(* LS Electric XG5000 project: XMC_SingleAxis_FBs *)
(* sample programs for single axis function blocks. *)
(* PLC LSPLC *)
(* module base 0 slot 0: Input/Output Module:XMC-DN24 (DC 24V Input 8Points/TR output 16Points) *)
(* module base 0 slot 1: Internal Analog Input/Output:XMF-AH04E (A/D voltage/current 2 channels, D/A voltage 2 channels) *)
(* task Periodic Task: Kind=2 *)
(* task Initialization Task: Kind=1 *)
(* task NC Program: Kind=6 *)
VAR_GLOBAL
    ContinuousRelative_INST : MC_MOVECONTINUOUSRELATIVE; (* MC_MoveContinuousRelative fb *)
    Relative_INST : MC_MOVECONTINUOUSRELATIVE; (* MC_MoveContinuousRelative fb *)
END_VAR

PROGRAM ECAT_Connect_Example (* task: Scan Program *)
VAR
    Connect_Error : BOOL; (* status that LS_Connect has an error *)
    Connect_ErrorID : WORD; (* LS_Connect Error number *)
    Connect_INST : LS_CONNECT; (* LS_Connect fb *)
    Disconnect_Error : BOOL; (* status that LS_Disconnect has an error *)
    Disconnect_ErrorID : WORD; (* Error Number for LS_Disconnect FB *)
    Disconnect_INST : LS_DISCONNECT; (* LS_Disconnect fb *)
    Execute_Connect : BOOL; (* Execute LS_Connect fb *)
    Execute_Disconnect : BOOL; (* execute LS_Disconnect fb *)
END_VAR

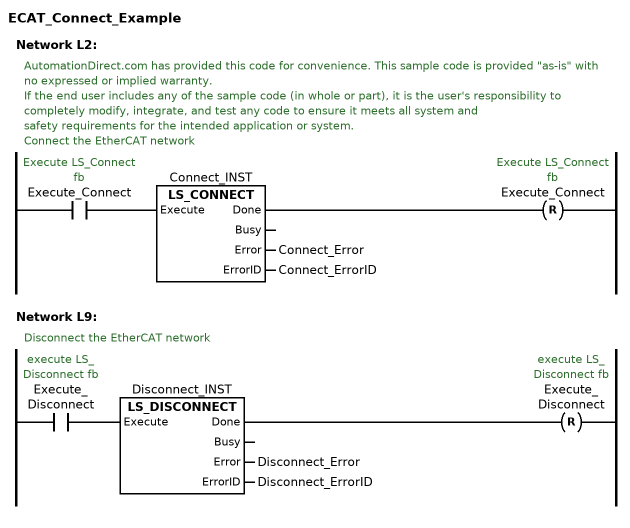
(* AutomationDirect.com has provided this code for convenience. This sample code is provided "as-is" with no expressed or implied warranty. / If the end user includes any of the sample code (in whole or part), it is the user's responsibility to completely modify, integrate, and test any code to ensure it meets all system and / safety requirements for the intended application or system. *)
(* Connect the EtherCAT network *)
(* Rung L2 *)
Connect_INST(Execute := Execute_Connect, Error => Connect_Error, ErrorID => Connect_ErrorID);
IF Connect_INST.Done THEN Execute_Connect := FALSE; END_IF;
(* Disconnect the EtherCAT network *)
(* Rung L9 *)
Disconnect_INST(Execute := Execute_Disconnect, Error => Disconnect_Error, ErrorID => Disconnect_ErrorID);
IF Disconnect_INST.Done THEN Execute_Disconnect := FALSE; END_IF;
END_PROGRAM

PROGRAM MC_Power_Example (* task: Scan Program *)
VAR
    Axis1 : UINT; (* used to tell MC function blocks to use axis 1 *)
    Axis1_MCPower_Error : BOOL; (* status of MC_Power error status *)
    Axis1_MCPower_ErrorID : WORD; (* error id of Axis 1 MC_Power *)
    Axis1_Power_Status : BOOL; (* status of axis 1 power *)
    Axis1_Power_Valid : BOOL; (* Axis1 power status is valid *)
    Power_INST : MC_POWER; (* MC_Power fb *)
    Power_On_Axis1 : BOOL; (* command to turn on power to axis 1 *)
END_VAR

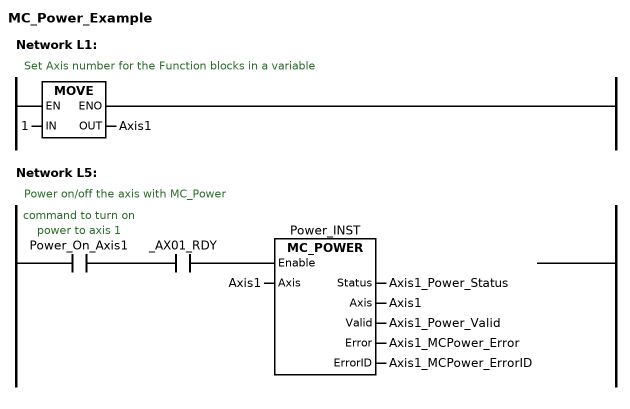
(* Set Axis number for the Function blocks in a variable *)
(* Rung L1 *)
Axis1 := 1;
(* Power on/off the axis with MC_Power *)
(* Rung L5 *)
Power_INST(Enable := Power_On_Axis1 AND _AX01_RDY, Axis := Axis1, Status => Axis1_Power_Status, Axis => Axis1, Valid => Axis1_Power_Valid, Error => Axis1_MCPower_Error, ErrorID => Axis1_MCPower_ErrorID);
END_PROGRAM

PROGRAM Home_Example (* task: Scan Program *)
(* example of MC_Home and LS_Home *)
VAR
    Axis1 : UINT; (* used to tell MC function blocks to use axis 1 *)
    Execute_LS_Home : BOOL; (* Execute LS_Home fb *)
    Execute_MC_Home : BOOL; (* execute MC_Home fb *)
    Home_INST : MC_HOME; (* MC_Home fb *)
    LSHome_Aborted : BOOL; (* LS_Home fb command aborted status *)
    LSHome_Active : BOOL; (* LS_Home fb active status *)
    LSHome_Busy : BOOL; (* LS_Home busy status *)
    LSHome_Error : BOOL; (* LSHome fb error status *)
    LSHome_ErrorID : WORD; (* LS_Home fb error id value *)
    LS_Home_INST : LS_HOME; (* LS_Home fb *)
    MCHome_Aborted : BOOL; (* MC_Home command was aborted *)
    MCHome_Active : BOOL; (* MC_Home is active *)
    MCHome_Busy : BOOL; (* MC_Home is busy *)
    MCHome_Error : BOOL; (* error status of MC_Home *)
    MCHome_ErrorID : WORD; (* error id value for MC_Home *)
END_VAR

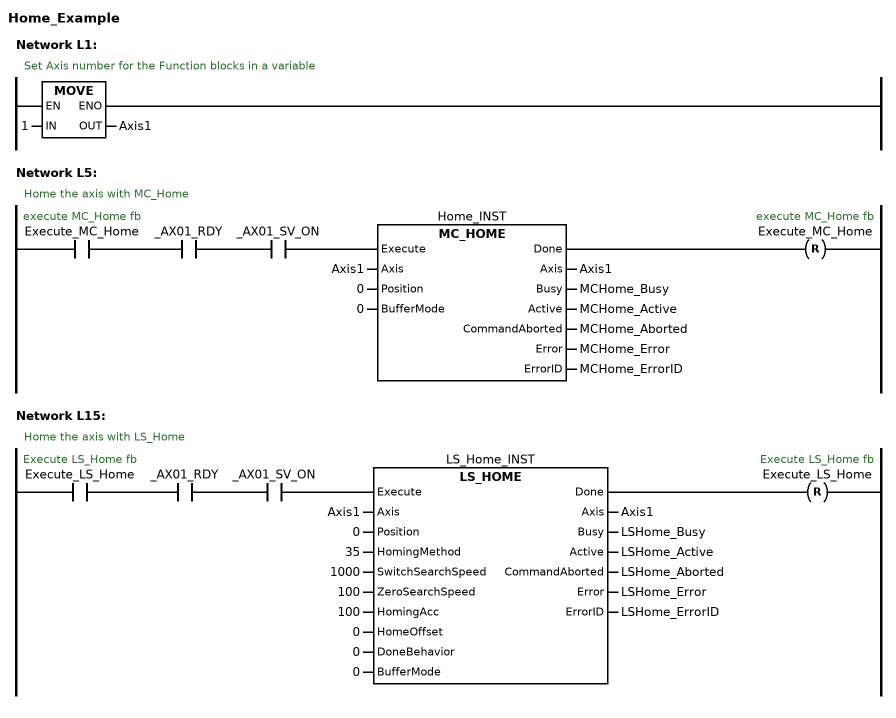
(* Set Axis number for the Function blocks in a variable *)
(* Rung L1 *)
Axis1 := 1;
(* Home the axis with MC_Home *)
(* Rung L5 *)
Home_INST(Execute := Execute_MC_Home AND _AX01_RDY AND _AX01_SV_ON, Axis := Axis1, Position := 0, BufferMode := 0, Axis => Axis1, Busy => MCHome_Busy, Active => MCHome_Active, CommandAborted => MCHome_Aborted, Error => MCHome_Error, ErrorID => MCHome_ErrorID);
IF Home_INST.Done THEN Execute_MC_Home := FALSE; END_IF;
(* Home the axis with LS_Home *)
(* Rung L15 *)
LS_Home_INST(Execute := Execute_LS_Home AND _AX01_RDY AND _AX01_SV_ON, Axis := Axis1, Position := 0, HomingMethod := 35, SwitchSearchSpeed := 1000, ZeroSearchSpeed := 100, HomingAcc := 100, HomeOffset := 0, DoneBehavior := 0, BufferMode := 0, Axis => Axis1, Busy => LSHome_Busy, Active => LSHome_Active, CommandAborted => LSHome_Aborted, Error => LSHome_Error, ErrorID => LSHome_ErrorID);
IF LS_Home_INST.Done THEN Execute_LS_Home := FALSE; END_IF;
END_PROGRAM

PROGRAM MCStop_MCHalt_Examples (* task: Scan Program *)
(* Examples of MC_Stop and MC_Hault function blocks. *)
VAR
    Axis1 : UINT; (* used to tell MC function blocks to use axis 1 *)
    Execute_MCHalt : BOOL; (* execute MC_Halt FB *)
    Execute_MCStop : BOOL; (* command to execute MC_Stop fb *)
    MCHalt_Aborted : BOOL; (* MC_Hault command aborted status *)
    MCHalt_Active : BOOL; (* MC_Halt active status *)
    MCHalt_Busy : BOOL; (* Busy status for MC_Halt *)
    MCHalt_Error : BOOL; (* MC_Halt error status *)
    MCHalt_ErrorID : WORD; (* MC_Halt Error identification value *)
    MCHalt_INST : MC_HALT; (* MC_Halt function block *)
    MCStop_Aborted : BOOL; (* MC_Stop aborted status *)
    MCStop_Busy : BOOL; (* MC_Stop Busy Status *)
    MCStop_Error : BOOL; (* MC_Stop error status *)
    MCStop_ErrorID : WORD; (* MC_Stop error identification value *)
    MCStop_INST : MC_STOP; (* MC_Stop function block *)
END_VAR

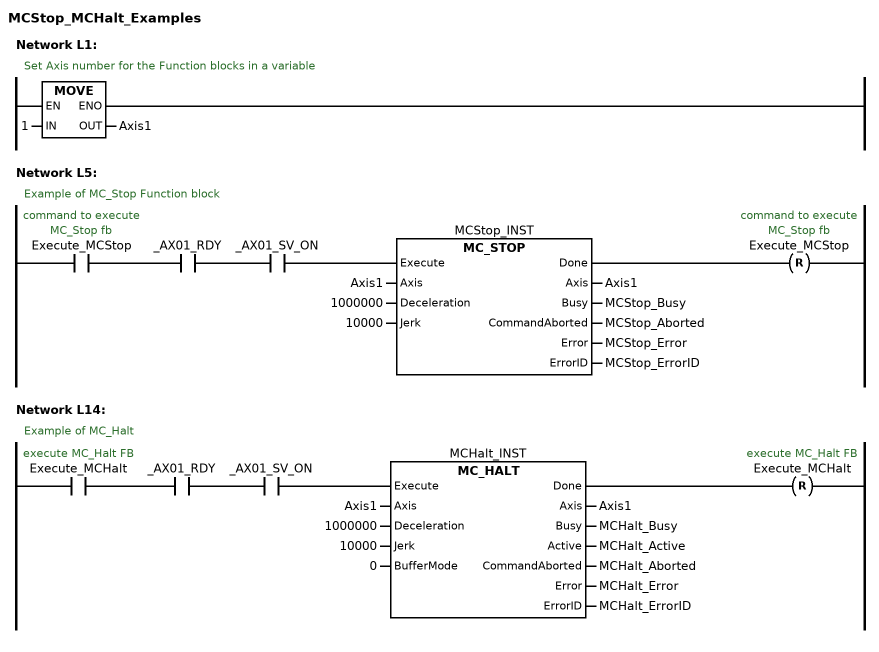
(* Set Axis number for the Function blocks in a variable *)
(* Rung L1 *)
Axis1 := 1;
(* Example of MC_Stop Function block *)
(* Rung L5 *)
MCStop_INST(Execute := Execute_MCStop AND _AX01_RDY AND _AX01_SV_ON, Axis := Axis1, Deceleration := 1000000, Jerk := 10000, Axis => Axis1, Busy => MCStop_Busy, CommandAborted => MCStop_Aborted, Error => MCStop_Error, ErrorID => MCStop_ErrorID);
IF MCStop_INST.Done THEN Execute_MCStop := FALSE; END_IF;
(* Example of MC_Halt *)
(* Rung L14 *)
MCHalt_INST(Execute := Execute_MCHalt AND _AX01_RDY AND _AX01_SV_ON, Axis := Axis1, Deceleration := 1000000, Jerk := 10000, BufferMode := 0, Axis => Axis1, Busy => MCHalt_Busy, Active => MCHalt_Active, CommandAborted => MCHalt_Aborted, Error => MCHalt_Error, ErrorID => MCHalt_ErrorID);
IF MCHalt_INST.Done THEN Execute_MCHalt := FALSE; END_IF;
END_PROGRAM

PROGRAM MC_ReadMotionInfo_Example (* task: Scan Program *)
(* example program for MC_ReadMotionInfo *)
VAR
    Axis1 : UINT; (* used to tell MC function blocks to use axis 1 *)
    Axis1_Info_Busy : BOOL; (* Axis 1 MC_ReadMotionInfo is busy *)
    Axis1_Info_Error : BOOL; (* Axis 1 MC_ReadMotionInfo error status *)
    Axis1_Info_ErrorID : WORD; (* Axis 1 MC_ReadMotionInfo error identfication *)
    Axis1_Info_Valid : BOOL; (* MC_ReadMotionInfo fb for axis 1 is valid *)
    Axis1_ParameterNumber : INT; (* Parameter number for MC_ReadMotionInfo *)
    Axis1_Value32 : REAL; (* Axis 1 MC_ReadMotionInfo Value32 outptut *)
    Axis1_Value64 : LREAL; (* Axis1 MC_ReadMotionInfo Value64 output *)
    MotionInfo_INST : MC_READMOTIONINFO; (* MC_ReadMotionInfo function block *)
    Read_Axis1_MotionInfo : BOOL; (* command to read axis 1 motion information *)
END_VAR

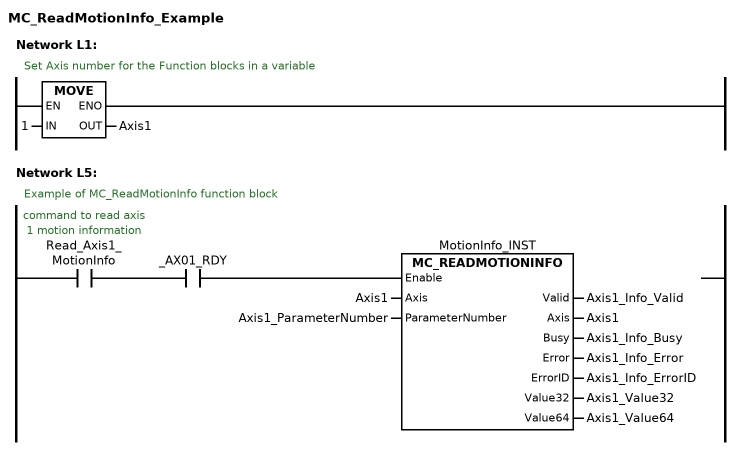
(* Set Axis number for the Function blocks in a variable *)
(* Rung L1 *)
Axis1 := 1;
(* Example of MC_ReadMotionInfo function block *)
(* Rung L5 *)
MotionInfo_INST(Enable := Read_Axis1_MotionInfo AND _AX01_RDY, Axis := Axis1, ParameterNumber := Axis1_ParameterNumber, Valid => Axis1_Info_Valid, Axis => Axis1, Busy => Axis1_Info_Busy, Error => Axis1_Info_Error, ErrorID => Axis1_Info_ErrorID, Value32 => Axis1_Value32, Value64 => Axis1_Value64);
END_PROGRAM

PROGRAM MC_ReadActualPosition_Example (* task: Scan Program *)
(* example program for MC_ReadActualPosition function block *)
VAR
    Axis1 : UINT; (* used to tell MC function blocks to use axis 1 *)
    Axis1_Position_Busy : BOOL; (* MC_ReadActualPosition is busy *)
    Axis1_Position_Error : BOOL; (* MC_ReadActualPosition error status *)
    Axis1_Position_ErrorID : WORD; (* MC_ReadActualPosition error identification *)
    Axis1_Position_Valid : BOOL; (* Axis 1 MC_ReadActualPosition value is valid *)
    Axis1_Position_Value32 : REAL; (* REAL value of Axis1 current position *)
    Axis1_Position_Value64 : LREAL; (* Axis 1 LREAL position value *)
    Axis1_Read_Position : BOOL; (* enable Axis1 MC_ReadActualPosition fb *)
    ReadPosition_INST : MC_READACTUALPOSITION; (* MC_ReadActualPosition function block *)
END_VAR

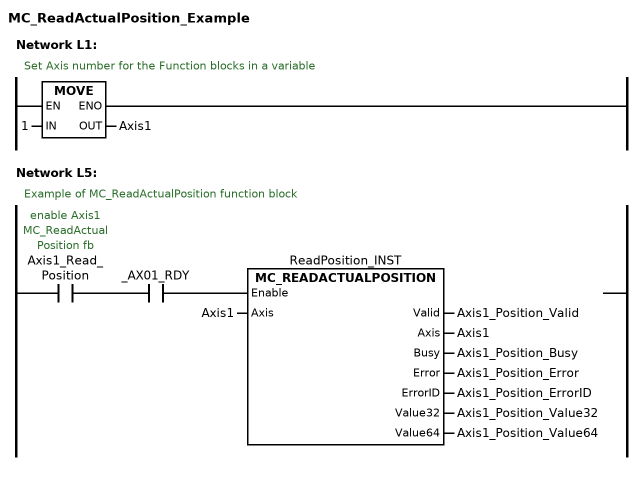
(* Set Axis number for the Function blocks in a variable *)
(* Rung L1 *)
Axis1 := 1;
(* Example of MC_ReadActualPosition function block *)
(* Rung L5 *)
ReadPosition_INST(Enable := Axis1_Read_Position AND _AX01_RDY, Axis := Axis1, Valid => Axis1_Position_Valid, Axis => Axis1, Busy => Axis1_Position_Busy, Error => Axis1_Position_Error, ErrorID => Axis1_Position_ErrorID, Value32 => Axis1_Position_Value32, Value64 => Axis1_Position_Value64);
END_PROGRAM

PROGRAM MC_ReadActualVelocity_Example (* task: Scan Program *)
(* example program for MC_ReadActualVelocity function block *)
VAR
    Axis1 : UINT; (* used to tell MC function blocks to use axis 1 *)
    Axis1_Read_Velocity : BOOL; (* command to enable MC_ReadActualVelocity *)
    Axis1_Velocity_Busy : BOOL; (* Axis 1 MC_ReadActualVelocity busy status *)
    Axis1_Velocity_Error : BOOL; (* Axis 1 MC_ReadActualVelocity error status *)
    Axis1_Velocity_ErrorID : WORD; (* Axis 1 MC_ReadActualVelocity error identification *)
    Axis1_Velocity_Valid : BOOL; (* Axis1 MC_ReadActualVelocity is valid *)
    Axis1_Velocity_Value32 : REAL; (* Axis 1 MC_ReadActualVelocity REAL value *)
    Axis1_Velocity_Value64 : LREAL; (* Axis1 MC_ReadActualVelocity LREAL value *)
    ReadVelocity_INST : MC_READACTUALVELOCITY; (* MC_ReadActualVelocity function block *)
END_VAR

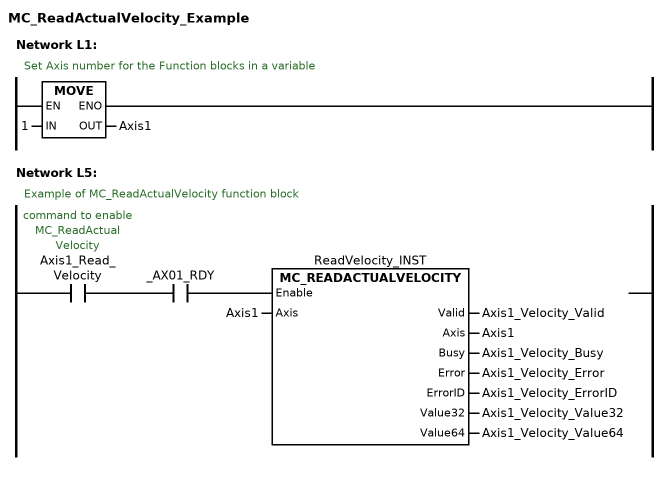
(* Set Axis number for the Function blocks in a variable *)
(* Rung L1 *)
Axis1 := 1;
(* Example of MC_ReadActualVelocity function block *)
(* Rung L5 *)
ReadVelocity_INST(Enable := Axis1_Read_Velocity AND _AX01_RDY, Axis := Axis1, Valid => Axis1_Velocity_Valid, Axis => Axis1, Busy => Axis1_Velocity_Busy, Error => Axis1_Velocity_Error, ErrorID => Axis1_Velocity_ErrorID, Value32 => Axis1_Velocity_Value32, Value64 => Axis1_Velocity_Value64);
END_PROGRAM

PROGRAM MC_ReadActualTorque_Example (* task: Scan Program *)
(* MC_ReadActualTorque function block example *)
VAR
    Axis1 : UINT; (* used to tell MC function blocks to use axis 1 *)
    Axis1_Read_Torque : BOOL; (* enable MC_ReadActualTorque *)
    Axis1_Torque_Busy : BOOL; (* Axis 1 MC_ReadActualTorque is busy *)
    Axis1_Torque_Error : BOOL; (* Axis1 MC_ReadActualTorque error status *)
    Axis1_Torque_ErrorID : WORD; (* Axis 1 MC_ReadActualTorque error identification *)
    Axis1_Torque_Valid : BOOL; (* Axis 1 MC_ReadActualTorque value is valid *)
    Axis1_Torque_Value32 : REAL; (* Axis 1 torque REAL value *)
    Axis1_Torque_Value64 : LREAL; (* Axis 1 torque LREAL value *)
    ReadTorque_INST : MC_READACTUALTORQUE; (* MC_ReadActualTorque function block *)
END_VAR

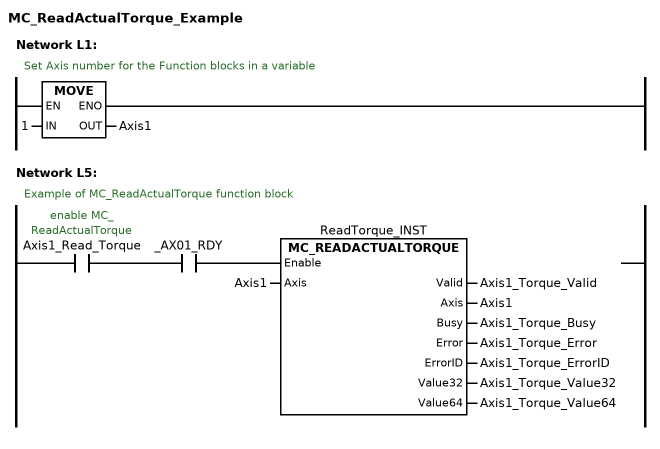
(* Set Axis number for the Function blocks in a variable *)
(* Rung L1 *)
Axis1 := 1;
(* Example of MC_ReadActualTorque function block *)
(* Rung L5 *)
ReadTorque_INST(Enable := Axis1_Read_Torque AND _AX01_RDY, Axis := Axis1, Valid => Axis1_Torque_Valid, Axis => Axis1, Busy => Axis1_Torque_Busy, Error => Axis1_Torque_Error, ErrorID => Axis1_Torque_ErrorID, Value32 => Axis1_Torque_Value32, Value64 => Axis1_Torque_Value64);
END_PROGRAM

PROGRAM MC_Reset_Example (* task: Scan Program *)
(* example of MC_Reset and MC_Reset2 function blocks. *)
VAR
    Axis1 : UINT; (* used to tell MC function blocks to use axis 1 *)
    Execute_MCReset : BOOL; (* command to execute MC_Reset FB. *)
    Execute_MCReset2 : BOOL; (* command to execute MC_Reset2 *)
    Reset1_Busy : BOOL; (* MC_Reset busy status *)
    Reset1_Error : BOOL; (* MC_Reset Error status *)
    Reset1_ErrorID : WORD; (* MC_Reset error identification *)
    Reset1_ErrorType : BOOL; (* error type for MC_Reset *)
    Reset1_INST : MC_RESET; (* MC_Reset function block *)
    Reset2_Busy : BOOL; (* busy status for MC_Reset2 *)
    Reset2_Error : BOOL; (* error status for MC_Reset2 *)
    Reset2_ErrorID : WORD; (* MC_Reset2 error identification *)
    Reset2_ErrorType : UINT; (* error type for MC_Reset2 *)
    Reset2_INST : MC_RESET2; (* MC_Reset2 function block *)
END_VAR

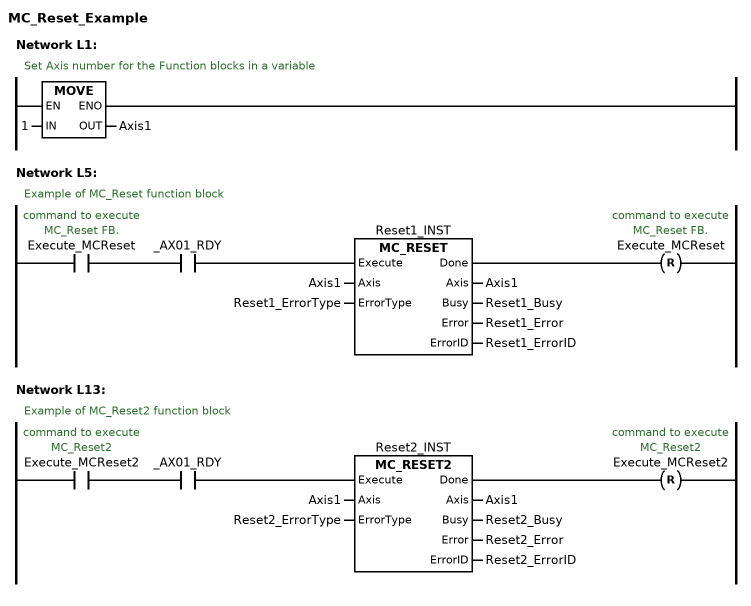
(* Set Axis number for the Function blocks in a variable *)
(* Rung L1 *)
Axis1 := 1;
(* Example of MC_Reset function block *)
(* Rung L5 *)
Reset1_INST(Execute := Execute_MCReset AND _AX01_RDY, Axis := Axis1, ErrorType := Reset1_ErrorType, Axis => Axis1, Busy => Reset1_Busy, Error => Reset1_Error, ErrorID => Reset1_ErrorID);
IF Reset1_INST.Done THEN Execute_MCReset := FALSE; END_IF;
(* Example of MC_Reset2 function block *)
(* Rung L13 *)
Reset2_INST(Execute := Execute_MCReset2 AND _AX01_RDY, Axis := Axis1, ErrorType := Reset2_ErrorType, Axis => Axis1, Busy => Reset2_Busy, Error => Reset2_Error, ErrorID => Reset2_ErrorID);
IF Reset2_INST.Done THEN Execute_MCReset2 := FALSE; END_IF;
END_PROGRAM

PROGRAM MC_MoveAbsolute_Example (* task: Scan Program *)
(* example program for MC_MoveAbsolute function block *)
VAR
    AbsoluteMove_Aborted : BOOL; (* MC_MoveAbsolute was aborted. *)
    AbsoluteMove_Acceleration : LREAL; (* acceleration for MC_MoveAbsolute *)
    AbsoluteMove_Active : BOOL; (* MC_MoveAbsolute is active *)
    AbsoluteMove_Busy : BOOL; (* MC_MoveAbsolute busy status *)
    AbsoluteMove_ContinuousUpdate : BOOL; (* continuous update status for MC_MoveAbsolute *)
    AbsoluteMove_Deceleration : LREAL; (* deceleration for MC_MoveAbsolute *)
    AbsoluteMove_Direction : UINT; (* direction of MC_MoveAbsolute *)
    AbsoluteMove_Error : BOOL; (* MC_MoveAbsolute error status *)
    AbsoluteMove_ErrorID : WORD; (* MC_MoveAbsolute error identification *)
    AbsoluteMove_Jerk : LREAL; (* jerk value for MC_MoveAbsolute *)
    AbsoluteMove_TargetPosition : LREAL; (* target position for MC_MoveAbsolute *)
    AbsoluteMove_Velocity : LREAL; (* velocity for MC_MoveAbsolute *)
    Absolute_INST : MC_MOVEABSOLUTE; (* MC_MoveAbsolute function block *)
    Axis1 : UINT; (* used to tell MC function blocks to use axis 1 *)
    Execute_Absolute_Move : BOOL; (* execute MC_MoveAbsolute function block *)
END_VAR

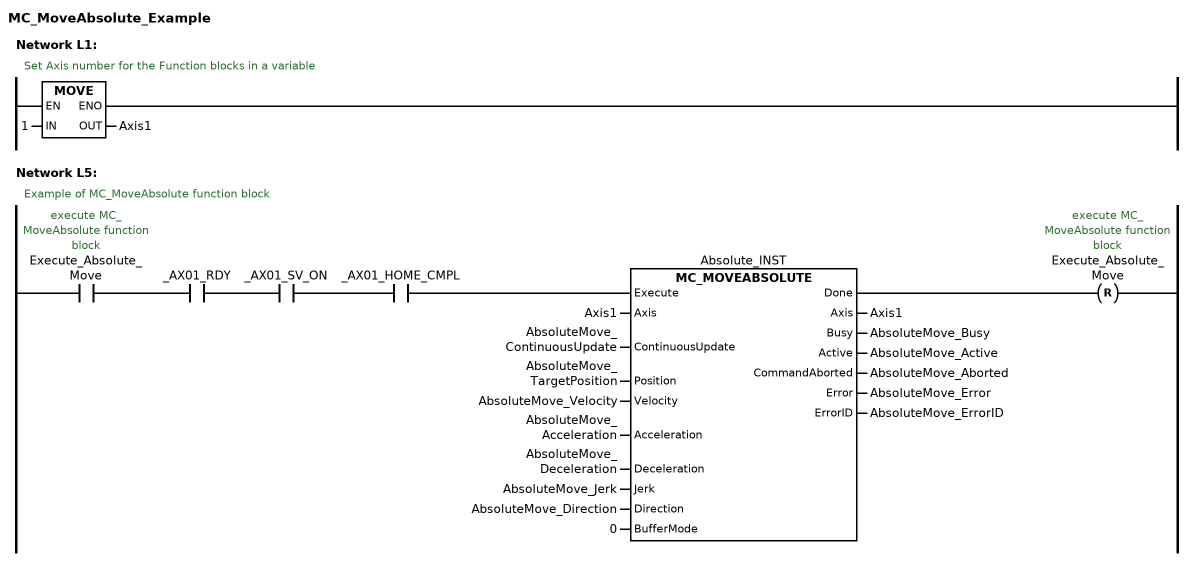
(* Set Axis number for the Function blocks in a variable *)
(* Rung L1 *)
Axis1 := 1;
(* Example of MC_MoveAbsolute function block *)
(* Rung L5 *)
Absolute_INST(Execute := Execute_Absolute_Move AND _AX01_RDY AND _AX01_SV_ON AND _AX01_HOME_CMPL, Axis := Axis1, ContinuousUpdate := AbsoluteMove_ContinuousUpdate, Position := AbsoluteMove_TargetPosition, Velocity := AbsoluteMove_Velocity, Acceleration := AbsoluteMove_Acceleration, Deceleration := AbsoluteMove_Deceleration, Jerk := AbsoluteMove_Jerk, Direction := AbsoluteMove_Direction, BufferMode := 0, Axis => Axis1, Busy => AbsoluteMove_Busy, Active => AbsoluteMove_Active, CommandAborted => AbsoluteMove_Aborted, Error => AbsoluteMove_Error, ErrorID => AbsoluteMove_ErrorID);
IF Absolute_INST.Done THEN Execute_Absolute_Move := FALSE; END_IF;
END_PROGRAM

PROGRAM MC_MoveRelative_Example (* task: Scan Program *)
(* example program for MC_MoveRelative funciton block *)
VAR
    Axis1 : UINT; (* used to tell MC function blocks to use axis 1 *)
    Execute_RelativeMove : BOOL; (* execute MC_MoveRelative *)
    RelativeMove_Aborted : BOOL; (* MC_MoveRelative aborted status *)
    RelativeMove_Acceleration : LREAL; (* acceleration for relative move *)
    RelativeMove_Active : BOOL; (* MC_MoveRelative active status *)
    RelativeMove_Busy : BOOL; (* MC_MoveRelative busy status *)
    RelativeMove_ContinuousUpdate : BOOL; (* MC_MoveRelative continuous update *)
    RelativeMove_Deceleration : LREAL; (* deceleration for relative move *)
    RelativeMove_Distance : LREAL; (* Distance for the MC_MoveRelative to move *)
    RelativeMove_Error : BOOL; (* MC_MoveRelative error status *)
    RelativeMove_ErrorID : WORD; (* MC_MoveRelative error identification *)
    RelativeMove_INST : MC_MOVERELATIVE; (* MC_MoveRelative function block *)
    RelativeMove_Jerk : LREAL; (* jerk value for relative move *)
    RelativeMove_Velocity : LREAL; (* velocity for relative move *)
END_VAR

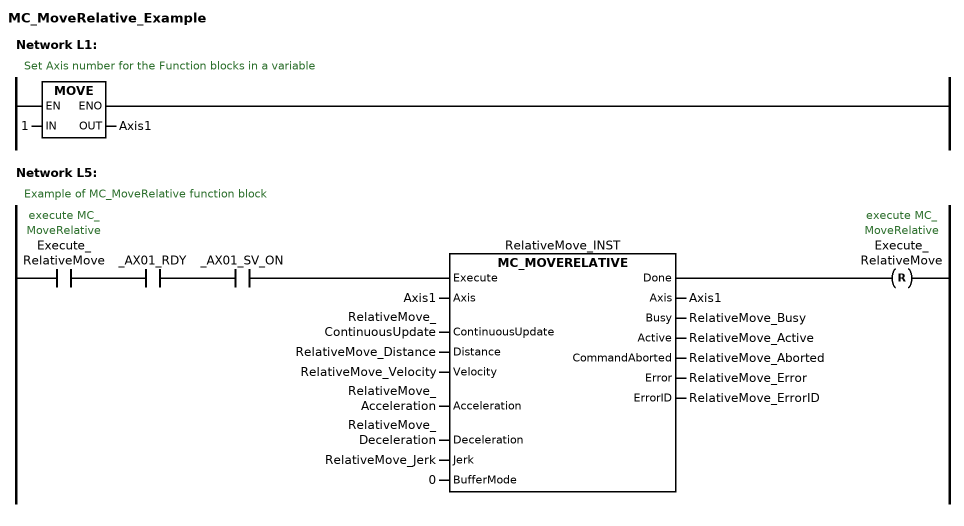
(* Set Axis number for the Function blocks in a variable *)
(* Rung L1 *)
Axis1 := 1;
(* Example of MC_MoveRelative function block *)
(* Rung L5 *)
RelativeMove_INST(Execute := Execute_RelativeMove AND _AX01_RDY AND _AX01_SV_ON, Axis := Axis1, ContinuousUpdate := RelativeMove_ContinuousUpdate, Distance := RelativeMove_Distance, Velocity := RelativeMove_Velocity, Acceleration := RelativeMove_Acceleration, Deceleration := RelativeMove_Deceleration, Jerk := RelativeMove_Jerk, BufferMode := 0, Axis => Axis1, Busy => RelativeMove_Busy, Active => RelativeMove_Active, CommandAborted => RelativeMove_Aborted, Error => RelativeMove_Error, ErrorID => RelativeMove_ErrorID);
IF RelativeMove_INST.Done THEN Execute_RelativeMove := FALSE; END_IF;
END_PROGRAM

PROGRAM MC_MoveAdditive_Example (* task: Scan Program *)
(* example program for MC_MoveAdditive *)
VAR
    AdditiveMove_Aborted : BOOL; (* MC_MoveAdditive aborted status *)
    AdditiveMove_Acceleration : LREAL; (* acceleration for MC_AdditiveMove *)
    AdditiveMove_Active : BOOL; (* MC_MoveAdditive active status *)
    AdditiveMove_Busy : BOOL; (* MC_MoveAdditive busy status *)
    AdditiveMove_ContinuousUpdate : BOOL; (* ContinuousUpdate for MC_MoveAdditive *)
    AdditiveMove_Deceleration : LREAL; (* deceleration for MC_AdditiveMove *)
    AdditiveMove_Distance : LREAL; (* distance for MC_MoveAdditive *)
    AdditiveMove_Error : BOOL; (* MC_MoveAdditive error status *)
    AdditiveMove_ErrorID : WORD; (* MC_MoveAdditive error identification *)
    AdditiveMove_INST : MC_MOVEADDITIVE; (* MC_MoveAdditive function block *)
    AdditiveMove_Jerk : LREAL; (* jerk value for MC_MoveAdditive *)
    AdditiveMove_Velocity : LREAL; (* velocity for the MC_MoveAdditive *)
    Axis1 : UINT; (* used to tell MC function blocks to use axis 1 *)
    Execute_AdditiveMove : BOOL; (* execute MC_MoveRelative *)
END_VAR

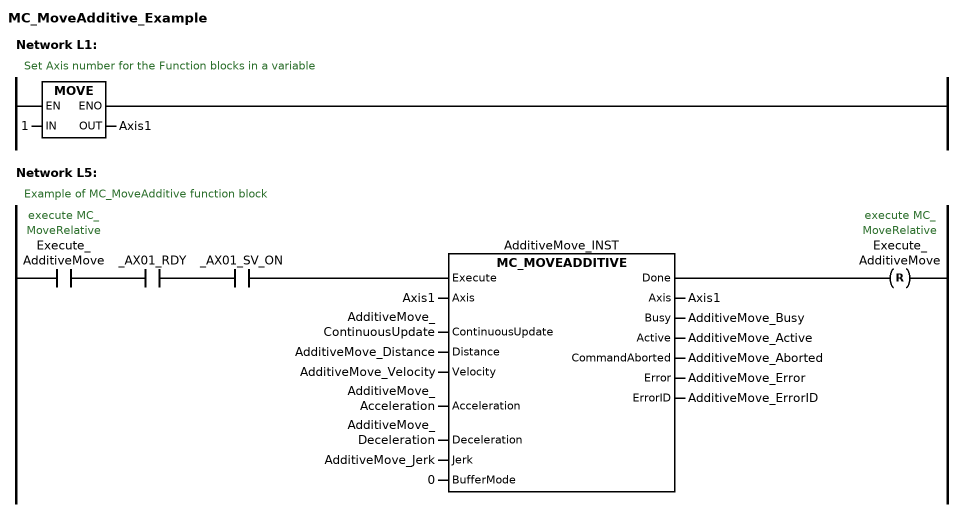
(* Set Axis number for the Function blocks in a variable *)
(* Rung L1 *)
Axis1 := 1;
(* Example of MC_MoveAdditive function block *)
(* Rung L5 *)
AdditiveMove_INST(Execute := Execute_AdditiveMove AND _AX01_RDY AND _AX01_SV_ON, Axis := Axis1, ContinuousUpdate := AdditiveMove_ContinuousUpdate, Distance := AdditiveMove_Distance, Velocity := AdditiveMove_Velocity, Acceleration := AdditiveMove_Acceleration, Deceleration := AdditiveMove_Deceleration, Jerk := AdditiveMove_Jerk, BufferMode := 0, Axis => Axis1, Busy => AdditiveMove_Busy, Active => AdditiveMove_Active, CommandAborted => AdditiveMove_Aborted, Error => AdditiveMove_Error, ErrorID => AdditiveMove_ErrorID);
IF AdditiveMove_INST.Done THEN Execute_AdditiveMove := FALSE; END_IF;
END_PROGRAM

PROGRAM MC_MoveVelocity_Example (* task: Scan Program *)
(* Example program for MC_MoveVelocity function block *)
VAR
    Axis1 : UINT; (* used to tell MC function blocks to use axis 1 *)
    Execute_MoveVelocity : BOOL; (* execute the MC_MoveVelocity Function block *)
    VelocityMove_Aborted : BOOL; (* MC_MoveVelocity Status aborted *)
    VelocityMove_Acceleration : LREAL; (* acceleration value for axis 1 MC_MoveVelocity *)
    VelocityMove_Active : BOOL; (* active status of MC_MoveVelocity *)
    VelocityMove_Busy : BOOL; (* busy status of MC_MoveVelocity *)
    VelocityMove_ContinuousUpdate : BOOL; (* setting the continuous update *)
    VelocityMove_Deceleration : LREAL; (* Axis1 deceleration value *)
    VelocityMove_Direction : UINT; (* direction of Axis 1 MC_MoveVelocity *)
    VelocityMove_Error : BOOL; (* Error status of MC_MoveVelocity *)
    VelocityMove_ErrorID : WORD; (* MC_MoveVelocity error identification *)
    VelocityMove_Jerk : LREAL; (* jerk value for axis 1 *)
    VelocityMove_Velocity : LREAL; (* velocity for Axis1 *)
    Velocity_INST : MC_MOVEVELOCITY; (* MC_MoveVelocity function block instance *)
END_VAR

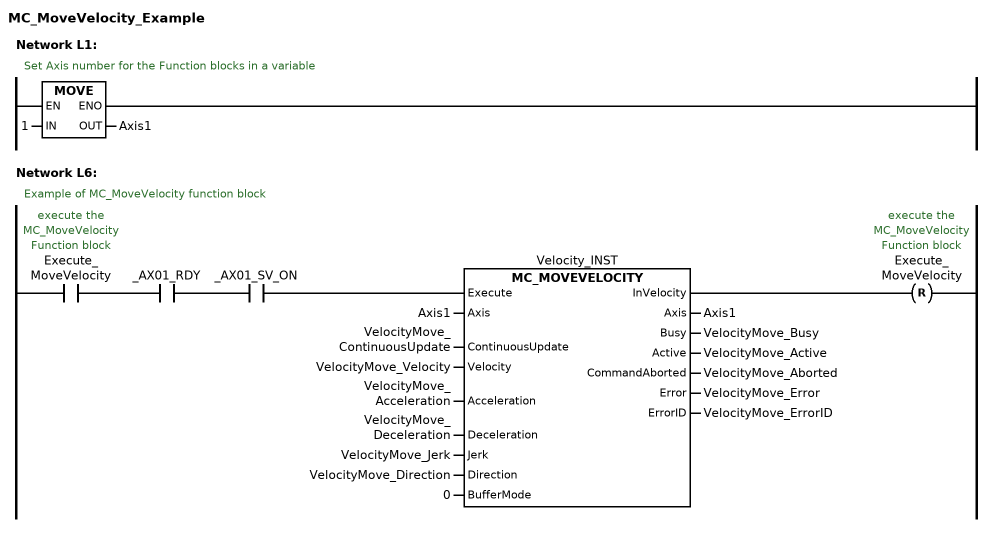
(* Set Axis number for the Function blocks in a variable *)
(* Rung L1 *)
Axis1 := 1;
(* Example of MC_MoveVelocity function block *)
(* Rung L6 *)
Velocity_INST(Execute := Execute_MoveVelocity AND _AX01_RDY AND _AX01_SV_ON, Axis := Axis1, ContinuousUpdate := VelocityMove_ContinuousUpdate, Velocity := VelocityMove_Velocity, Acceleration := VelocityMove_Acceleration, Deceleration := VelocityMove_Deceleration, Jerk := VelocityMove_Jerk, Direction := VelocityMove_Direction, BufferMode := 0, Axis => Axis1, Busy => VelocityMove_Busy, Active => VelocityMove_Active, CommandAborted => VelocityMove_Aborted, Error => VelocityMove_Error, ErrorID => VelocityMove_ErrorID);
IF Velocity_INST.InVelocity THEN Execute_MoveVelocity := FALSE; END_IF;
END_PROGRAM

PROGRAM MC_MoveContinuousAbsolute_Example (* task: Scan Program *)
(* example program for MC_MoveContinuousAbsolute function block *)
VAR
    Axis1 : UINT; (* used to tell MC function blocks to use axis 1 *)
    ContinuousAbsolute_Aborted : BOOL; (* aborted status of the function block *)
    ContinuousAbsolute_Acceleration : LREAL; (* acceleration for movement *)
    ContinuousAbsolute_Active : BOOL; (* active status of function block *)
    ContinuousAbsolute_Busy : BOOL; (* busy status *)
    ContinuousAbsolute_ContinuousUpdate : BOOL; (* MC_MoveContinuousAbsolute continuous update input *)
    ContinuousAbsolute_Deceleration : LREAL; (* deceleration for moves *)
    ContinuousAbsolute_Direction : UINT; (* direction of the movement *)
    ContinuousAbsolute_EndVelocity : LREAL; (* end velocity for MC_MoveContinuousAbsolute function block *)
    ContinuousAbsolute_Error : BOOL; (* error status of the function block *)
    ContinuousAbsolute_ErrorID : WORD; (* error identification of the function block *)
    ContinuousAbsolute_INST : MC_MOVECONTINUOUSABSOLUTE; (* MC_MoveContinuousAbsolute function block *)
    ContinuousAbsolute_Jerk : LREAL; (* jerk value for movement *)
    ContinuousAbsolute_Position : LREAL; (* target position before continuous motion *)
    ContinuousAbsolute_Velocity : LREAL; (* velocity of the absolute motion portion *)
    Execute_MoveContinuousAbsolute : BOOL; (* execute MC_MoveContinuousAbsolute *)
END_VAR

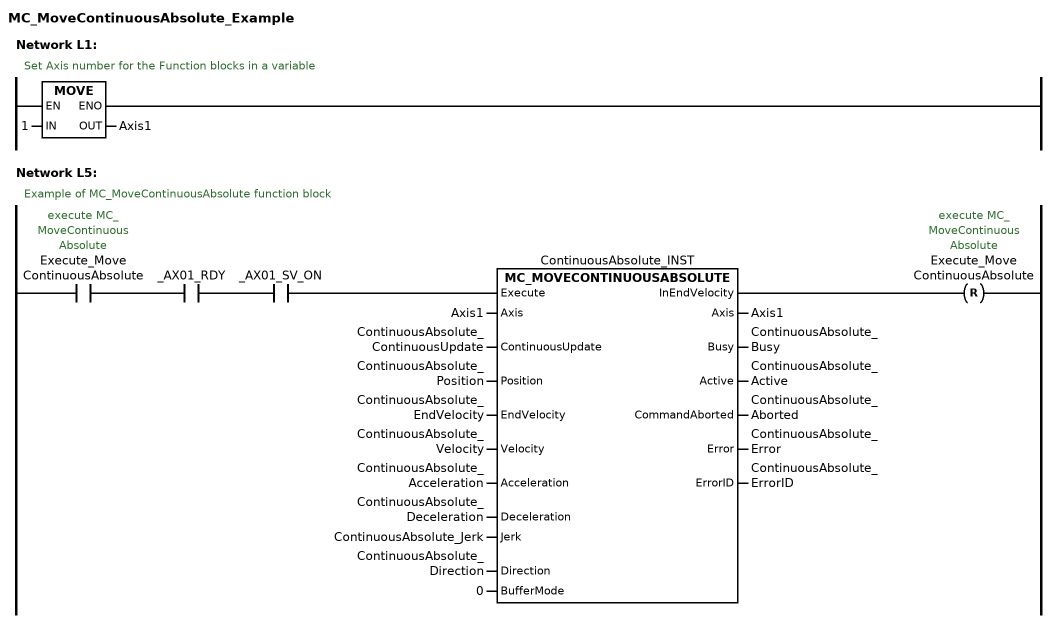
(* Set Axis number for the Function blocks in a variable *)
(* Rung L1 *)
Axis1 := 1;
(* Example of MC_MoveContinuousAbsolute function block *)
(* Rung L5 *)
ContinuousAbsolute_INST(Execute := Execute_MoveContinuousAbsolute AND _AX01_RDY AND _AX01_SV_ON, Axis := Axis1, ContinuousUpdate := ContinuousAbsolute_ContinuousUpdate, Position := ContinuousAbsolute_Position, EndVelocity := ContinuousAbsolute_EndVelocity, Velocity := ContinuousAbsolute_Velocity, Acceleration := ContinuousAbsolute_Acceleration, Deceleration := ContinuousAbsolute_Deceleration, Jerk := ContinuousAbsolute_Jerk, Direction := ContinuousAbsolute_Direction, BufferMode := 0, Axis => Axis1, Busy => ContinuousAbsolute_Busy, Active => ContinuousAbsolute_Active, CommandAborted => ContinuousAbsolute_Aborted, Error => ContinuousAbsolute_Error, ErrorID => ContinuousAbsolute_ErrorID);
IF ContinuousAbsolute_INST.InEndVelocity THEN Execute_MoveContinuousAbsolute := FALSE; END_IF;
END_PROGRAM

PROGRAM MC_MoveContinuousRelative_Example (* task: Scan Program *)
(* example of MC_MoveContinuousRelative function block *)
VAR
    Axis1 : UINT; (* used to tell MC function blocks to use axis 1 *)
    ContinuousRelative_Aborted : BOOL; (* aborted status for fb *)
    ContinuousRelative_Acceleration : LREAL; (* Acceleration for fb *)
    ContinuousRelative_Active : BOOL; (* active status for fb *)
    ContinuousRelative_Busy : BOOL; (* busy status for fb *)
    ContinuousRelative_ContinuousUpdate : BOOL; (* MC_MoveContinuousRelative update input *)
    ContinuousRelative_Deceleration : LREAL; (* deceleration for fb *)
    ContinuousRelative_Distance : LREAL; (* distance value for MC_MoveContinuousRelative *)
    ContinuousRelative_EndVelocity : LREAL; (* end velocity value for MC_MoveContinuousRelative fb *)
    ContinuousRelative_Error : BOOL; (* error status for fb *)
    ContinuousRelative_ErrorID : WORD; (* error identification for fb *)
    ContinuousRelative_Jerk : LREAL; (* Jerk value for fb *)
    ContinuousRelative_Velocity : LREAL; (* Relative move velocity for MC_MoveContinuousRelative *)
    Execute_ContinuousRelative : BOOL; (* command to execute MC_MoveContinuousRelative fb *)
END_VAR
VAR_EXTERNAL
    ContinuousRelative_INST : MC_MOVECONTINUOUSRELATIVE; (* MC_MoveContinuousRelative fb *)
END_VAR

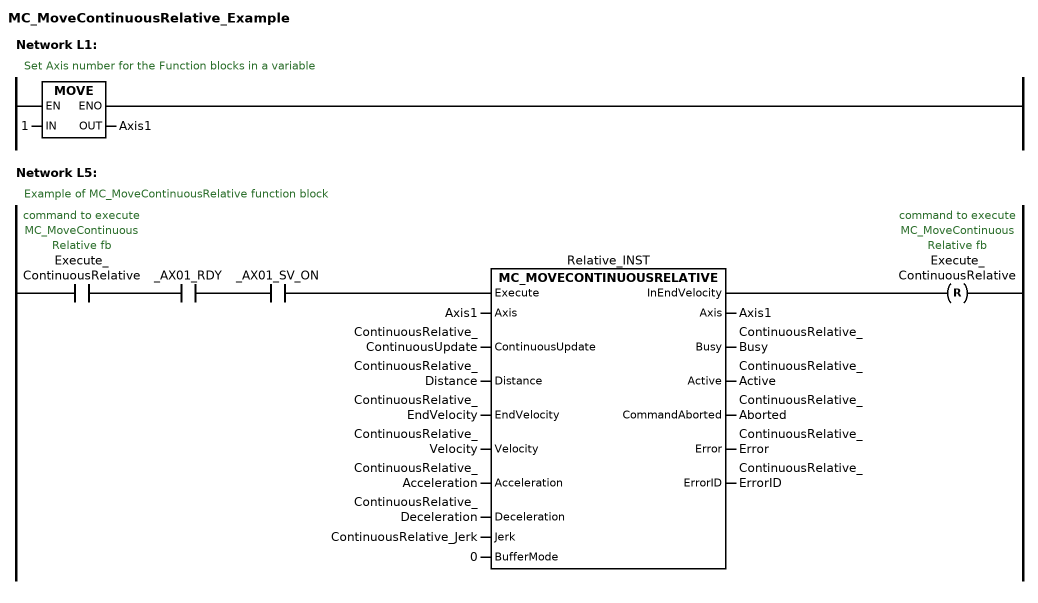
(* Set Axis number for the Function blocks in a variable *)
(* Rung L1 *)
Axis1 := 1;
(* Example of MC_MoveContinuousRelative function block *)
(* Rung L5 *)
Relative_INST(Execute := Execute_ContinuousRelative AND _AX01_RDY AND _AX01_SV_ON, Axis := Axis1, ContinuousUpdate := ContinuousRelative_ContinuousUpdate, Distance := ContinuousRelative_Distance, EndVelocity := ContinuousRelative_EndVelocity, Velocity := ContinuousRelative_Velocity, Acceleration := ContinuousRelative_Acceleration, Deceleration := ContinuousRelative_Deceleration, Jerk := ContinuousRelative_Jerk, BufferMode := 0, Axis => Axis1, Busy => ContinuousRelative_Busy, Active => ContinuousRelative_Active, CommandAborted => ContinuousRelative_Aborted, Error => ContinuousRelative_Error, ErrorID => ContinuousRelative_ErrorID);
IF Relative_INST.InEndVelocity THEN Execute_ContinuousRelative := FALSE; END_IF;
END_PROGRAM

PROGRAM MC_TorqueControl_Example (* task: Scan Program *)
(* example program for MC_TorqueControl *)
VAR
    Axis1 : UINT; (* used to tell MC function blocks to use axis 1 *)
    ContinuousUpdate : BOOL; (* continuous update of TorqueControl *)
    Execute_Torque_Control : BOOL; (* execute MC_TorqueControl function block *)
    TorqueControl_Aborted : BOOL; (* torque control aborted status *)
    TorqueControl_Active : BOOL; (* torque control active status *)
    TorqueControl_BufferMode : UINT; (* Buffer Mode for Axis 1 MC_TorqueControl *)
    TorqueControl_Busy : BOOL; (* torque control busy status *)
    TorqueControl_Direction : UINT; (* Axis1 direction for MC_TorqueControl *)
    TorqueControl_Error : BOOL; (* torque control error status *)
    TorqueControl_ErrorID : WORD; (* torque control error identification *)
    TorqueControl_TorqueRamp : LREAL; (* torque Ramp for axis 1 *)
    TorqueControl_TorqueValue : LREAL; (* torque value for axis 1 MC_TorqueControl *)
    Torque_Ctrl_INST : MC_TORQUECONTROL; (* MC_TorqueControl function block *)
END_VAR

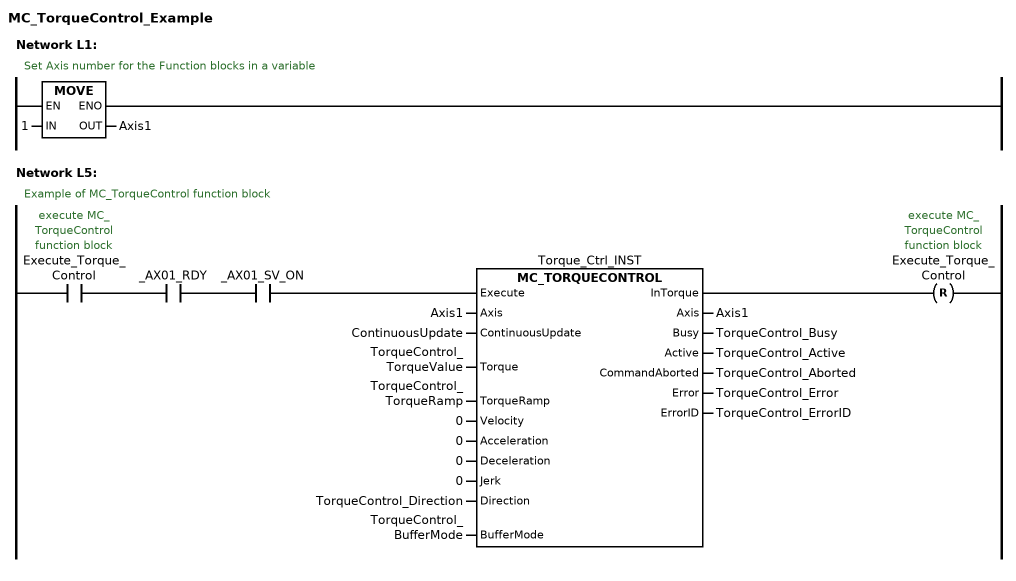
(* Set Axis number for the Function blocks in a variable *)
(* Rung L1 *)
Axis1 := 1;
(* Example of MC_TorqueControl function block *)
(* Rung L5 *)
Torque_Ctrl_INST(Execute := Execute_Torque_Control AND _AX01_RDY AND _AX01_SV_ON, Axis := Axis1, ContinuousUpdate := ContinuousUpdate, Torque := TorqueControl_TorqueValue, TorqueRamp := TorqueControl_TorqueRamp, Velocity := 0, Acceleration := 0, Deceleration := 0, Jerk := 0, Direction := TorqueControl_Direction, BufferMode := TorqueControl_BufferMode, Axis => Axis1, Busy => TorqueControl_Busy, Active => TorqueControl_Active, CommandAborted => TorqueControl_Aborted, Error => TorqueControl_Error, ErrorID => TorqueControl_ErrorID);
IF Torque_Ctrl_INST.InTorque THEN Execute_Torque_Control := FALSE; END_IF;
END_PROGRAM

PROGRAM MC_SetPosition_Example (* task: Scan Program *)
(* example of MC_SetPosition function block *)
VAR
    Axis1 : UINT; (* used to tell MC function blocks to use axis 1 *)
    Execute_Set_Position : BOOL; (* execute the MC_SetPosition FB *)
    SetPosition_Aborted : BOOL; (* aborted status of MC_SetPosition *)
    SetPosition_Busy : BOOL; (* busy status of MC_SetPosition *)
    SetPosition_Error : BOOL; (* Error status of fb *)
    SetPosition_ErrorID : WORD; (* error identification of fb *)
    SetPosition_INST : MC_SETPOSITION; (* MC_SetPosition function block *)
    SetPosition_Position : LREAL; (* position value for set position *)
END_VAR

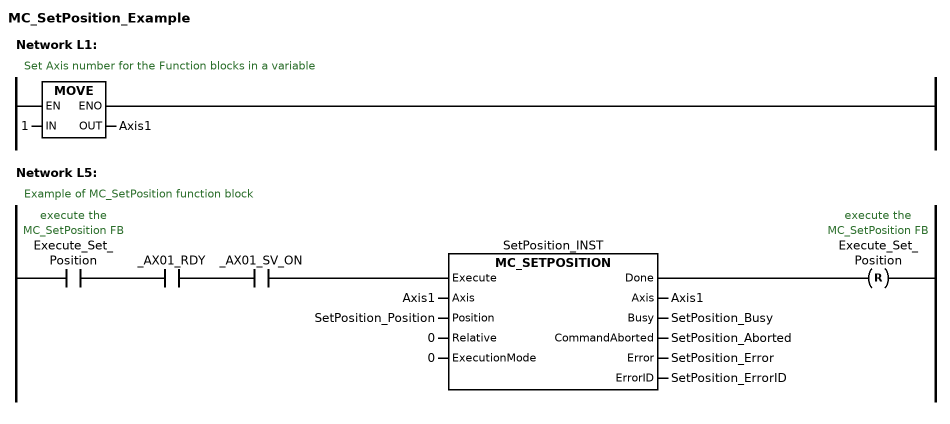
(* Set Axis number for the Function blocks in a variable *)
(* Rung L1 *)
Axis1 := 1;
(* Example of MC_SetPosition function block *)
(* Rung L5 *)
SetPosition_INST(Execute := Execute_Set_Position AND _AX01_RDY AND _AX01_SV_ON, Axis := Axis1, Position := SetPosition_Position, Relative := 0, ExecutionMode := 0, Axis => Axis1, Busy => SetPosition_Busy, CommandAborted => SetPosition_Aborted, Error => SetPosition_Error, ErrorID => SetPosition_ErrorID);
IF SetPosition_INST.Done THEN Execute_Set_Position := FALSE; END_IF;
END_PROGRAM

PROGRAM MC_SetOverride_Example (* task: Scan Program *)
(* example program for MC_SetOverride function block. *)
VAR
    Axis1 : UINT; (* used to tell MC function blocks to use axis 1 *)
    Execute_Speed_Override : BOOL; (* execute the MC_SetOverride fb *)
    Override_AccFactor : LREAL; (* override acceleration factor *)
    Override_Busy : BOOL; (* fb is busy *)
    Override_Enabled : BOOL; (* fb is enabled *)
    Override_Error : BOOL; (* fb error status *)
    Override_ErrorID : WORD; (* error identification for fb *)
    Override_INST : MC_SETOVERRIDE; (* MC_SetOverride function block *)
    Override_JerkFactor : LREAL; (* override jerk factor *)
    Override_VelFactor : LREAL; (* velocity override factor *)
END_VAR

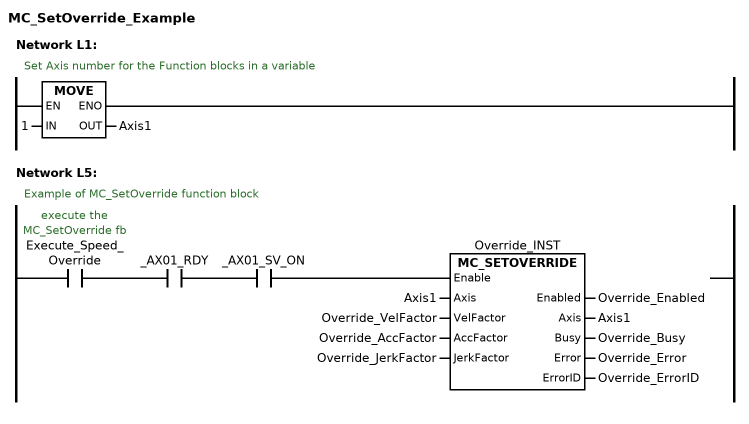
(* Set Axis number for the Function blocks in a variable *)
(* Rung L1 *)
Axis1 := 1;
(* Example of MC_SetOverride function block *)
(* Rung L5 *)
Override_INST(Enable := Execute_Speed_Override AND _AX01_RDY AND _AX01_SV_ON, Axis := Axis1, VelFactor := Override_VelFactor, AccFactor := Override_AccFactor, JerkFactor := Override_JerkFactor, Enabled => Override_Enabled, Axis => Axis1, Busy => Override_Busy, Error => Override_Error, ErrorID => Override_ErrorID);
END_PROGRAM

PROGRAM MC_ReadParameter_Example (* task: Scan Program *)
(* example program for MC_ReadParameter fb *)
VAR
    Axis1 : UINT; (* used to tell MC function blocks to use axis 1 *)
    Execute_Parameter_Read : BOOL; (* execute the MC_ReadParameter fb *)
    ParameterNumber : INT; (* parameter number to read *)
    ReadParam_Busy : BOOL; (* read parameter fb is busy *)
    ReadParam_Error : BOOL; (* error status of read parameter fb *)
    ReadParam_ErrorID : WORD; (* error identification for read parameter fb *)
    ReadParam_INST : MC_READPARAMETER; (* MC_ReadParameter function block *)
    ReadParam_Valid : BOOL; (* value for read parameter is valid *)
    ReadParam_Value : LREAL; (* value of parameter to read *)
END_VAR

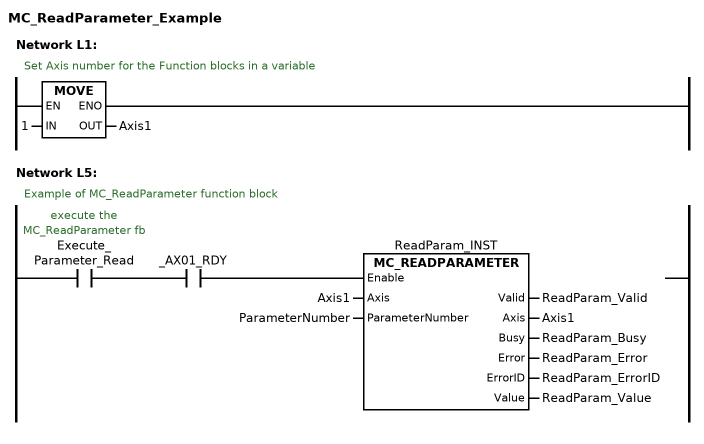
(* Set Axis number for the Function blocks in a variable *)
(* Rung L1 *)
Axis1 := 1;
(* Example of MC_ReadParameter function block *)
(* Rung L5 *)
ReadParam_INST(Enable := Execute_Parameter_Read AND _AX01_RDY, Axis := Axis1, ParameterNumber := ParameterNumber, Valid => ReadParam_Valid, Axis => Axis1, Busy => ReadParam_Busy, Error => ReadParam_Error, ErrorID => ReadParam_ErrorID, Value => ReadParam_Value);
END_PROGRAM

PROGRAM MC_WriteParameter_Example (* task: Scan Program *)
(* example of MC_WriteParameter function block *)
VAR
    Axis1 : UINT; (* used to tell MC function blocks to use axis 1 *)
    Execute_Write_Parameter : BOOL; (* execute the MC_WriteParameter fb *)
    ParameterNumber : INT; (* parameter to write to *)
    WriteParam_Busy : BOOL; (* busy status *)
    WriteParam_Error : BOOL; (* error status *)
    WriteParam_ErrorID : WORD; (* error identification *)
    WriteParam_INST : MC_WRITEPARAMETER; (* MC_WriteParameter function block *)
    WriteParam_Value : LREAL; (* value to write to the parameter *)
END_VAR

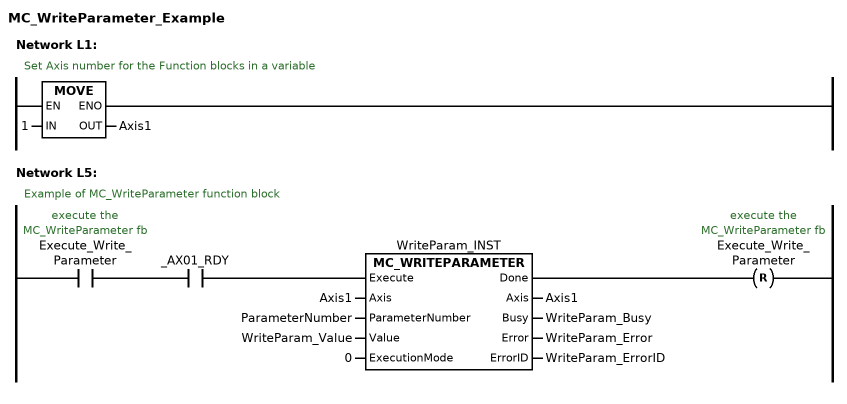
(* Set Axis number for the Function blocks in a variable *)
(* Rung L1 *)
Axis1 := 1;
(* Example of MC_WriteParameter function block *)
(* Rung L5 *)
WriteParam_INST(Execute := Execute_Write_Parameter AND _AX01_RDY, Axis := Axis1, ParameterNumber := ParameterNumber, Value := WriteParam_Value, ExecutionMode := 0, Axis => Axis1, Busy => WriteParam_Busy, Error => WriteParam_Error, ErrorID => WriteParam_ErrorID);
IF WriteParam_INST.Done THEN Execute_Write_Parameter := FALSE; END_IF;
END_PROGRAM

PROGRAM MC_TouchProbe&Ex_Example (* task: Scan Program *)
(* example program for MC_TouchProbe and MC_TouchProbeEx function blocks *)
VAR
    Axis1 : UINT; (* used to tell MC function blocks to use axis 1 *)
    Execute_TouchProbe : BOOL; (* execute the MC_TouchProbe function block *)
    Execute_TouchProbeEx : BOOL; (* execute MC_TouchProbeEx function block *)
    ProbeEx_Aborted : BOOL; (* aborted status for MC_TouchProbeEx *)
    ProbeEx_Busy : BOOL; (* busy status for MC_TouchProbeEx *)
    ProbeEx_Error : BOOL; (* error status for MC_TouchProbeEx *)
    ProbeEx_ErrorID : WORD; (* Error identification for MC_TouchProbeEx *)
    ProbeEx_INST : MC_TOUCHPROBEEX; (* MC_TouchProbeEx function block *)
    ProbeEx_RecordedPosition : LREAL; (* Recorded position for MC_TouchProbeEx *)
    ProbeEx_TriggerInput : UINT; (* TriggerInput for MC_TouchProbeEx *)
    ProbeEx_TriggerMode : UINT; (* Trigger mode for MC_TouchProbeEx *)
    Probe_Aborted : BOOL; (* Aborted status of MC_TouchProbe *)
    Probe_Busy : BOOL; (* busy status for MC_TouchProbe *)
    Probe_Error : BOOL; (* error status of MC_TouchProbe *)
    Probe_ErrorID : WORD; (* Error identification for MC_TouchProbe *)
    Probe_RecordedPosition : LREAL; (* recorded position for MC_TouchProbe *)
    Probe_TriggerInput : UINT; (* trigger input for MC_TouchProbe *)
    TouchProbe_INST : MC_TOUCHPROBE; (* MC_TouchProbe function block. *)
END_VAR

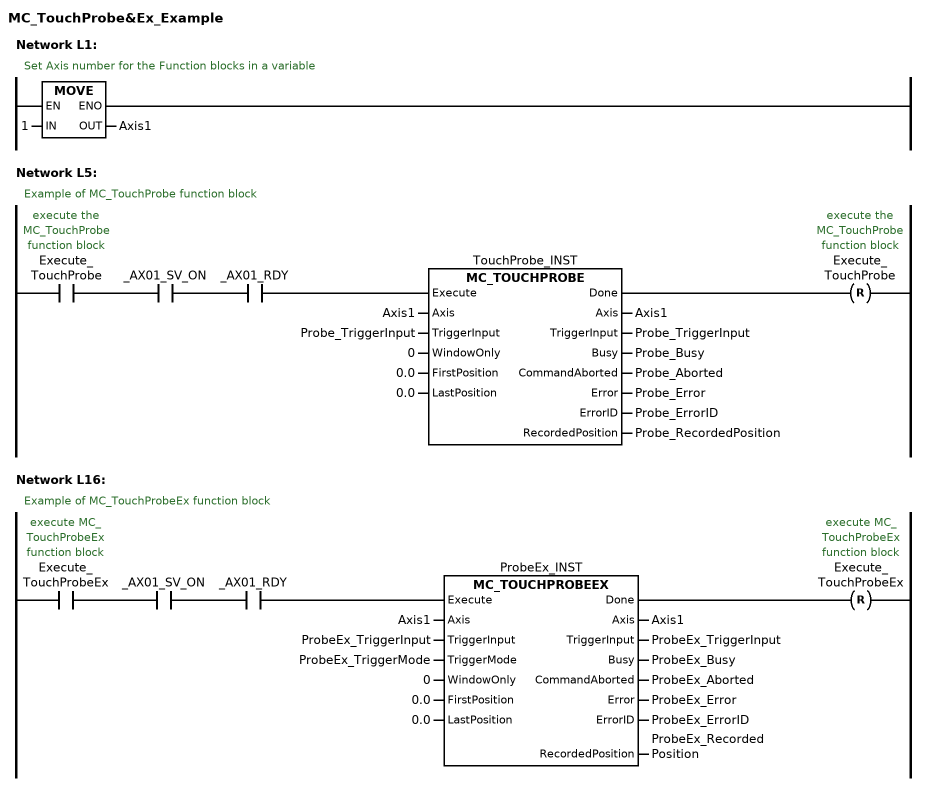
(* Set Axis number for the Function blocks in a variable *)
(* Rung L1 *)
Axis1 := 1;
(* Example of MC_TouchProbe function block *)
(* Rung L5 *)
TouchProbe_INST(Execute := Execute_TouchProbe AND _AX01_SV_ON AND _AX01_RDY, Axis := Axis1, TriggerInput := Probe_TriggerInput, WindowOnly := 0, FirstPosition := 0.0, LastPosition := 0.0, Axis => Axis1, TriggerInput => Probe_TriggerInput, Busy => Probe_Busy, CommandAborted => Probe_Aborted, Error => Probe_Error, ErrorID => Probe_ErrorID, RecordedPosition => Probe_RecordedPosition);
IF TouchProbe_INST.Done THEN Execute_TouchProbe := FALSE; END_IF;
(* Example of MC_TouchProbeEx function block *)
(* Rung L16 *)
ProbeEx_INST(Execute := Execute_TouchProbeEx AND _AX01_SV_ON AND _AX01_RDY, Axis := Axis1, TriggerInput := ProbeEx_TriggerInput, TriggerMode := ProbeEx_TriggerMode, WindowOnly := 0, FirstPosition := 0.0, LastPosition := 0.0, Axis => Axis1, TriggerInput => ProbeEx_TriggerInput, Busy => ProbeEx_Busy, CommandAborted => ProbeEx_Aborted, Error => ProbeEx_Error, ErrorID => ProbeEx_ErrorID, RecordedPosition => ProbeEx_RecordedPosition);
IF ProbeEx_INST.Done THEN Execute_TouchProbeEx := FALSE; END_IF;
END_PROGRAM

PROGRAM MC_AbortTrigger_Example (* task: Scan Program *)
(* example program for MC_AbortTrigger *)
VAR
    AbortTrigger_INST : MC_ABORTTRIGGER; (* MC_AbortTrigger Function block *)
    Abort_Busy : BOOL; (* MC_AbortTrigger busy status *)
    Abort_Error : BOOL; (* MC_AbortTrigger error status *)
    Abort_ErrorID : WORD; (* MC_AbortTrigger error identification *)
    Abort_TriggerInput : UINT; (* Trigger Input for MC_AbortTrigger *)
    Axis1 : UINT; (* used to tell MC function blocks to use axis 1 *)
    Execute_AbortTrigger : BOOL; (* execute MC_AbortTrigger *)
END_VAR

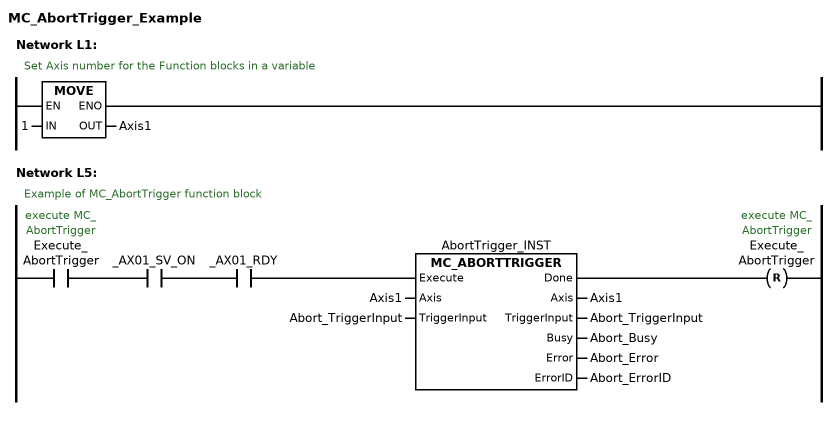
(* Set Axis number for the Function blocks in a variable *)
(* Rung L1 *)
Axis1 := 1;
(* Example of MC_AbortTrigger function block *)
(* Rung L5 *)
AbortTrigger_INST(Execute := Execute_AbortTrigger AND _AX01_SV_ON AND _AX01_RDY, Axis := Axis1, TriggerInput := Abort_TriggerInput, Axis => Axis1, TriggerInput => Abort_TriggerInput, Busy => Abort_Busy, Error => Abort_Error, ErrorID => Abort_ErrorID);
IF AbortTrigger_INST.Done THEN Execute_AbortTrigger := FALSE; END_IF;
END_PROGRAM

PROGRAM MC_SuperImposed_Example (* task: Scan Program *)
(* example for MC_SuperImposed and MC_HaltSuperImposed function blocks *)
VAR
    Axis1 : UINT; (* used to tell MC function blocks to use axis 1 *)
    Execute_HaltSuperImposed : BOOL; (* Halt super imposed movement *)
    Execute_SuperImposed : BOOL; (* execute the MC_MoveSuperImposed fb *)
    HaltImposed_Aborted : BOOL; (* command aborted status of MC_HaltSuperImposed *)
    HaltImposed_Busy : BOOL; (* busy status of MC_HaltSuperImposed *)
    HaltImposed_Deceleration : LREAL; (* deceleration of MC_HaltSuperImposed *)
    HaltImposed_Error : BOOL; (* error status of MC_HaltSuperImposed *)
    HaltImposed_ErrorID : WORD; (* error identification for MC_HaltSuperImposed *)
    HaltImposed_INST : MC_HALTSUPERIMPOSED; (* MC_HaltSuperImposed function block *)
    HaltImposed_Jerk : LREAL; (* MC_HaltSuperImposed jerk value *)
    SuperImposed_Aborted : BOOL; (* command aborted status for MC_MoveSuperImposed *)
    SuperImposed_Acceleration : LREAL; (* acceleration for MC_MoveSuperImposed *)
    SuperImposed_Active : BOOL; (* active status for MC_MoveSuperImposed *)
    SuperImposed_Busy : BOOL; (* busy status for MC_MoveSuperImposed *)
    SuperImposed_ContinuousUpdate : BOOL; (* continuous update input of MC_MoveSuperImposed *)
    SuperImposed_CoveredDistance : LREAL; (* distance covered by MC_MoveSuperImposed *)
    SuperImposed_Deceleration : LREAL; (* Deceleration for MC_MoveSuperImposed *)
    SuperImposed_Distance : LREAL; (* Distance for MC_MoveSuperImposed *)
    SuperImposed_Error : BOOL; (* error status for MC_MoveSuperImposed *)
    SuperImposed_ErrorID : WORD; (* error identification for MC_MoveSuperImposed *)
    SuperImposed_INST : MC_MOVESUPERIMPOSED; (* MC_MoveSuperImposed fb *)
    SuperImposed_Jerk : LREAL; (* jerk value for MC_MoveSuperImposed *)
    SuperImposed_VelocityDiff : LREAL; (* velocity difference for MC_MoveSuperImposed *)
END_VAR

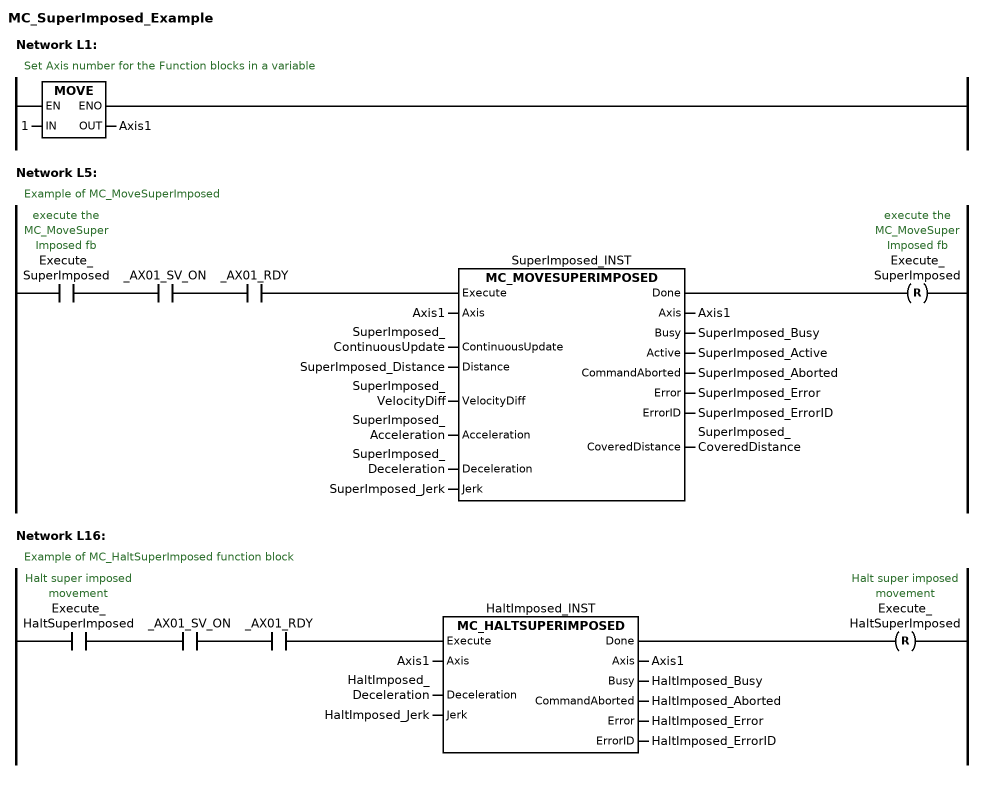
(* Set Axis number for the Function blocks in a variable *)
(* Rung L1 *)
Axis1 := 1;
(* Example of MC_MoveSuperImposed *)
(* Rung L5 *)
SuperImposed_INST(Execute := Execute_SuperImposed AND _AX01_SV_ON AND _AX01_RDY, Axis := Axis1, ContinuousUpdate := SuperImposed_ContinuousUpdate, Distance := SuperImposed_Distance, VelocityDiff := SuperImposed_VelocityDiff, Acceleration := SuperImposed_Acceleration, Deceleration := SuperImposed_Deceleration, Jerk := SuperImposed_Jerk, Axis => Axis1, Busy => SuperImposed_Busy, Active => SuperImposed_Active, CommandAborted => SuperImposed_Aborted, Error => SuperImposed_Error, ErrorID => SuperImposed_ErrorID, CoveredDistance => SuperImposed_CoveredDistance);
IF SuperImposed_INST.Done THEN Execute_SuperImposed := FALSE; END_IF;
(* Example of MC_HaltSuperImposed function block *)
(* Rung L16 *)
HaltImposed_INST(Execute := Execute_HaltSuperImposed AND _AX01_SV_ON AND _AX01_RDY, Axis := Axis1, Deceleration := HaltImposed_Deceleration, Jerk := HaltImposed_Jerk, Axis => Axis1, Busy => HaltImposed_Busy, CommandAborted => HaltImposed_Aborted, Error => HaltImposed_Error, ErrorID => HaltImposed_ErrorID);
IF HaltImposed_INST.Done THEN Execute_HaltSuperImposed := FALSE; END_IF;
END_PROGRAM

PROGRAM MC_ReadCommandedPosition_Example (* task: Scan Program *)
(* example program for MC_ReadCommandedPosition *)
VAR
    Axis1 : UINT; (* used to tell MC function blocks to use axis 1 *)
    Execute_ReadPosition : BOOL; (* enable MC_ReadCommandedPosition fb *)
    ReadPosition_Busy : BOOL; (* busy status for MC_ReadCommandedPosition *)
    ReadPosition_Error : BOOL; (* error status for MC_ReadCommandedPosition *)
    ReadPosition_ErrorID : WORD; (* error identification for MC_ReadCommandedPosition *)
    ReadPosition_INST : MC_READCOMMANDEDPOSITION; (* MC_ReadCommandedPosition function block *)
    ReadPosition_Valid : BOOL; (* MC_ReadCommandedPosition outputs are valid *)
    ReadPosition_Value32 : REAL; (* 32-bit position *)
    ReadPosition_Value64 : LREAL; (* 64-bit position *)
END_VAR

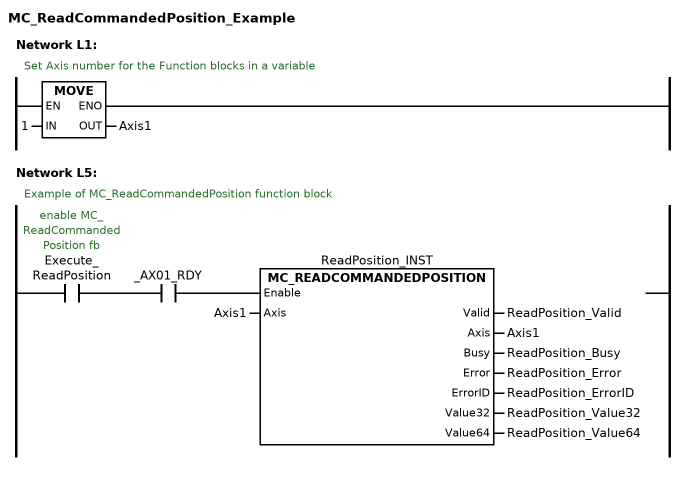
(* Set Axis number for the Function blocks in a variable *)
(* Rung L1 *)
Axis1 := 1;
(* Example of MC_ReadCommandedPosition function block *)
(* Rung L5 *)
ReadPosition_INST(Enable := Execute_ReadPosition AND _AX01_RDY, Axis := Axis1, Valid => ReadPosition_Valid, Axis => Axis1, Busy => ReadPosition_Busy, Error => ReadPosition_Error, ErrorID => ReadPosition_ErrorID, Value32 => ReadPosition_Value32, Value64 => ReadPosition_Value64);
END_PROGRAM

PROGRAM MC_ReadCommandedVelocity_Example (* task: Scan Program *)
(* example of MC_ReadCommandedVelocity fb *)
VAR
    Axis1 : UINT; (* used to tell MC function blocks to use axis 1 *)
    Execute_ReadVelocity : BOOL; (* enable the MC_ReadCommandedVelocity *)
    ReadVelocity_Busy : BOOL; (* busy status for MC_ReadCommandedVelocity *)
    ReadVelocity_Error : BOOL; (* error status for MC_ReadCommandedVelocity *)
    ReadVelocity_ErrorID : WORD; (* error identification for MC_ReadCommandedVelocity *)
    ReadVelocity_INST : MC_READCOMMANDEDVELOCITY; (* MC_ReadCommandedVelocity function block *)
    ReadVelocity_Valid : BOOL; (* MC_ReadCommandVelocity function block *)
    ReadVelocity_Value32 : REAL; (* REAL value for commanded velocity *)
    ReadVelocity_Value64 : LREAL; (* LREAL value for commanded velocity *)
END_VAR

